TYPE DUT_HMI_02_MANUALS :
STRUCT
	PS : ARRAY[0..CNC.NUM_MAX_MANUALS_02-1] OF BOOL;
	LS : ARRAY[0..CNC.NUM_MAX_MANUALS_02-1] OF BOOL;
END_STRUCT
END_TYPE

(* stored: Version 1.1.0.1, ProductVersion 3.1.4024.13
   DUT DUT_HMI_02_MANUALS: Id {a0ef8bb2-b95a-4fb6-b27a-879acba3f115} *)
